// TIA Portal project "E02_Timer" (V18)

(* hardware
DEVICE "S71500/ET200MP station_1"  S7-1500 station
   slot 0: "Telaio di montaggio_0"  Rack  6ES7 590-1***0-0AA0
   slot 1: "PLC_1"  CPU 1516-3 PN/DP  6ES7 516-3AN01-0AB0  V2.5
      slot 3: "Display CPU_1"  6ES7591-1BA00-0AA0
   slot 2: "DI 32x24VDC HF_1"  DI 32x24VDC HF  6ES7 521-1BL00-0AB0  V2.1
   slot 3: "DQ 32x24VDC/0.5A HF_1"  DQ 32x24VDC/0.5A HF  6ES7 522-1BL01-0AB0  V1.0
   slot 4: "AI 8xU/I/RTD/TC ST_1"  AI 8xU/I/RTD/TC ST  6ES7 531-7KF00-0AB0  V2.1
   slot 5: "AQ 4xU/I ST_1"  AQ 4xU/I ST  6ES7 532-5HD00-0AB0  V2.1
*)

// ===== PLC "PLC_1"  CPU 1516-3 PN/DP =====

VAR_GLOBAL   // PLC tag table "Tabella delle variabili standard"
   "Led1" AT %Q3.0 : Bool;
   "Led2" AT %Q3.1 : Bool;
   "Led3" AT %Q3.2 : Bool;
   "Led4" AT %Q3.3 : Bool;
   "Led5" AT %Q3.4 : Bool;
   "Led6" AT %Q3.5 : Bool;
   "Led7" AT %Q3.6 : Bool;
   "Led8" AT %Q3.7 : Bool;
END_VAR

DATA_BLOCK "DB_Comandi"   // DB1
{ S7_Optimized_Access := 'TRUE' }
VERSION : 0.1
   VAR
      btnStart : Bool;
      btnStop : Bool;
   END_VAR
BEGIN
END_DATA_BLOCK

DATA_BLOCK "DB_Variabili"   // DB2
{ S7_Optimized_Access := 'TRUE' }
VERSION : 0.1
   VAR
      Led1 : Bool;   // Variabili duplicate per sicurezza, non è quindi obbligatorio
      Led2 : Bool;
      Led3 : Bool;
      Led4 : Bool;
      Led5 : Bool;
      Led6 : Bool;
      Led7 : Bool;
      Led8 : Bool;
      TimerLampeggioSTART : Bool;
      TimerLampeggioDONE : Bool;
      TimerLampeggioOUTPUT : Time;
      TimerLampeggioDURATION : Time;
      inEsecuzione : Bool;
   END_VAR
BEGIN
END_DATA_BLOCK

// folder: System blocks/Program resources

DATA_BLOCK "TimerLampeggio"   // DB3
{ S7_Optimized_Access := 'TRUE' }
AUTHOR : Simatic
FAMILY : IEC
NAME : IEC_TMR
VERSION : 1.0
// stored: InstanceOfName IEC_TIMER
"IEC_TIMER"
BEGIN
END_DATA_BLOCK

// folder: (top level)

FUNCTION "FC_Grafcet" : Void   // FC1, SCL
{ S7_Optimized_Access := 'TRUE' }
VERSION : 0.1
BEGIN
   //Contiene il programma vero e proprio, codifica del "flow chart"
   //Se premo start avvio il timer
   //
   IF "DB_Comandi".btnStart = TRUE THEN
       "DB_Variabili".inEsecuzione := TRUE;
       "DB_Comandi".btnStart := FALSE;
   END_IF;
   //Se premo stop avvio il timer
   //
   IF "DB_Comandi".btnStop = TRUE THEN
       "DB_Variabili".inEsecuzione := FALSE;
       "DB_Comandi".btnStop := FALSE;
   END_IF;

   //Il funzionamento del timer dipende dalla variabile inEsecuzione e non dai 2 btn
   //
   IF "DB_Variabili".inEsecuzione = TRUE THEN
       "DB_Variabili".TimerLampeggioSTART := TRUE; //IL TIMER INIZIA A CONTARE
   ELSE
       "DB_Variabili".TimerLampeggioSTART := FALSE; //IL TIMER SI ARRESTA
   END_IF;

   //Gestisco il DONE del timer
   //
   IF "DB_Variabili".TimerLampeggioDONE = TRUE AND "DB_Variabili".inEsecuzione = TRUE THEN
       //Il timer ha contato fino alla fine
       //E voglio riprendere il ciclo dall'inizio
       "DB_Variabili".TimerLampeggioDONE := FALSE;
       "DB_Variabili".TimerLampeggioSTART := FALSE;
       //Accendo-spengo le uscite
       //
       "DB_Variabili".Led1 := NOT "DB_Variabili".Led1;
       "DB_Variabili".Led2 := NOT "DB_Variabili".Led2;
   END_IF;
END_FUNCTION

FUNCTION "FC_Timer" : Void   // FC2, SCL
{ S7_Optimized_Access := 'TRUE' }
VERSION : 0.1
BEGIN
   //Imposto la durata del timer
   "DB_Variabili".TimerLampeggioDURATION := T#5s;
   //

   "TimerLampeggio".TON(IN:="DB_Variabili".TimerLampeggioSTART, //Bool, portato a true fa partire il conteggio
                        PT:="DB_Variabili".TimerLampeggioDURATION, //Time, dice per quanto tempo deve contare
                        Q=>"DB_Variabili".TimerLampeggioDONE, //Quando Q = 1 (DONE), il conteggio è finito
                        ET=>"DB_Variabili".TimerLampeggioOUTPUT); //Visualizza il conteggio
END_FUNCTION

FUNCTION "FC_Uscite" : Void   // FC3, SCL
{ S7_Optimized_Access := 'TRUE' }
VERSION : 0.1
BEGIN
   //Fatto per sicurezza, controllo nuovamente che tutte le condizioni siano verificate
   //Scrivo fisicamente le uscite, dopo aver controllato che tutte le condizioni siano verificate

   "Led1" := "DB_Variabili".Led1;
   "Led2" := "DB_Variabili".Led2;
END_FUNCTION

ORGANIZATION_BLOCK "Main"   // OB1, LAD, ProgramCycle
TITLE = "Main Program Sweep (Cycle)"
{ S7_Optimized_Access := 'TRUE' }
VERSION : 0.1
   VAR_INPUT
      Initial_Call : Bool;   // Initial call of this OB
      Remanence : Bool;   // =True, if remanent data are available
   END_VAR
   VAR_TEMP   // added for the SCL form of the ladder/FBD networks
      _w1 : Bool;
      _w2 : Bool;
   END_VAR
BEGIN

REGION Network 1
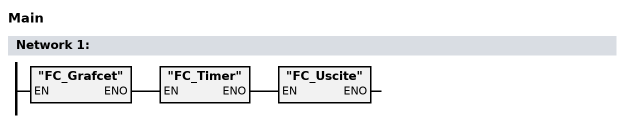
   RUNG wire#powerrail
      "FC_Grafcet"()
      "FC_Timer"()
      "FC_Uscite"()
   END_RUNG
   // the same network as SCL:
   "FC_Grafcet"(ENO => #_w1);
   "FC_Timer"(EN := #_w1, ENO => #_w2);
   IF #_w2 THEN "FC_Uscite"(); END_IF;
END_REGION
END_ORGANIZATION_BLOCK